// TIA Portal V18 export
VAR_GLOBAL   // PLC tag table "MES_NGCode"
END_VAR
VAR_GLOBAL CONSTANT   // user constants
   MES_NGCodeNG_Press : Int := 201;
   MES_NGCodeOK : Int := 0;
   MES_NGCodeIDIE : Int := 0;
   MES_NGCodeNG_illegal : Int := 201;
   MES_NGCodeNG_Manual : Int := 209;
END_VAR
